Staubli VAL3: RobotStatusMsg.pjx

--- RobotStatusMsg.pjx ---
Parameters version=s7.7.2 stackSize=5000 millimeterUnit=true
Program file=start.pgx
Program file=stop.pgx
Data file=RobotStatusMsg.dtx
Type name=RobotStatus path=Disk://RobotStatus/RobotStatus.pjx
Type name=Prefix path=Disk://Prefix/Prefix.pjx
Type name=Header path=Disk://Header/Header.pjx
Type name=Body path=Disk://Body/Body.pjx

--- RobotStatusMsg.dtx ---
public Body body
  [0]
    num nData[28]
public Header header
  [0]
    num nMsgType
    num nCommType
    num nReplyCode
    num nData[12]
public Prefix prefix
  [0]
    num nLength
    num nData[4]
public RobotStatus robotStatus
  [0]
    num nDrivesPowered
    num nEStopped
    num nErrorCode
    num nInError
    num nInMotion
    num nMode
    num nMotionPossible
